FUNCTION F_GET_TIME_STAMP : STRING(255)
VAR_INPUT
	systemTime				: TIMESTRUCT;			// Using Tc2_Utilities to have the TIMESTRUCT
	strSeparatorDate		: STRING(1) := '_';		// Separator between Year,Month,Day
	strSeparatorTime		: STRING(1) := ':';		// Separator between Hours, Minutes, Seconds		
END_VAR
VAR
	stYear					: STRING;
	stMonth					: STRING;
	stDay					: STRING;
	stHours					: STRING;
	stMinutes				: STRING;
	stSeconds				: STRING;
END_VAR

stYear 		:= CONCAT(WORD_TO_STRING(systemTime.wYear), strSeparatorDate);
stMonth		:= CONCAT(WORD_TO_STRING(systemTime.wMonth), strSeparatorDate);
stDay 		:= CONCAT(WORD_TO_STRING(systemTime.wDay), strSeparatorDate);
stHours 	:= CONCAT(WORD_TO_STRING(systemTime.wHour), strSeparatorTime);
stMinutes 	:= CONCAT(WORD_TO_STRING(systemTime.wMinute), strSeparatorTime);
stSeconds 	:= WORD_TO_STRING(systemTime.wSecond);
F_GET_TIME_STAMP := CONCAT(stYear,CONCAT(stMonth,CONCAT(stDay,CONCAT(stHours,CONCAT(stMinutes,stSeconds)))));

END_FUNCTION

(* stored: Version 1.1.0.1, ProductVersion 3.1.4024.9
   POU F_GET_TIME_STAMP: Id {9dd17d6a-0ac2-4820-8e12-49aeb4e7bd36}, SpecialFunc None *)
